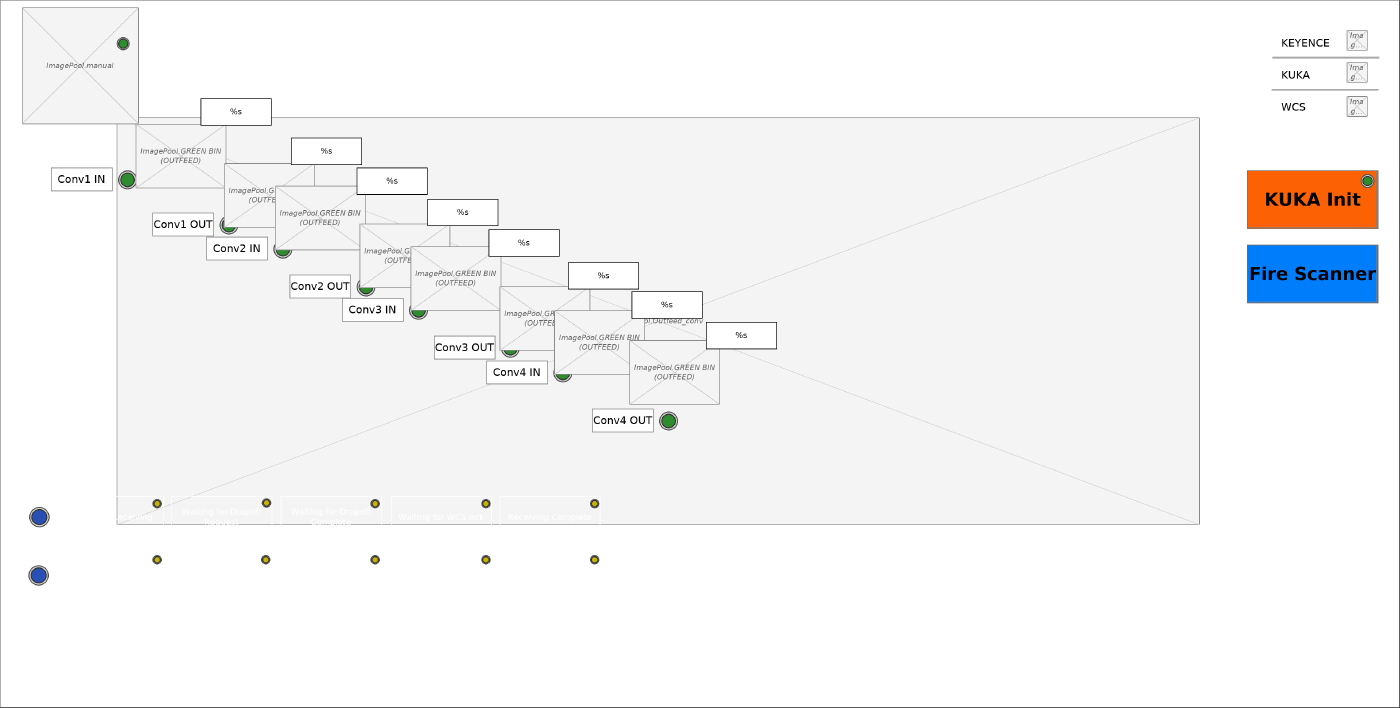
VISUALIZATION MAIN_CONTENT  // 1920x972
    Rectangle (0,0 1920x972)
    Image (160,161 1485x559), image: ImagePool.Outfeed_conv
    Group (1731,29 160x145)
        RoundedRectangle (0,0 160x145)
        RoundedRectangle (23,21 109x18), "KEYENCE"
        RoundedRectangle (23,65 92x18), "KUKA"
        RoundedRectangle (23,109 92x18), "WCS"
        Rectangle (14,49 146x2)
        Rectangle (13,93 146x2)
        Image (116,12 28x28), invisible if: IO.fbClient_QR.bConnected, image: ImagePool.no-wifi
        Image (116,12 28x28), invisible if: NOT IO.fbClient_QR.bConnected, image: ImagePool.wifi
        Image (116,56 28x28), invisible if: IO_KUKA.bPro_act, image: ImagePool.no-wifi
        Image (116,56 28x28), invisible if: NOT IO_KUKA.bPro_act, image: ImagePool.wifi
        Image (116,103 28x28), invisible if: IO.fbClient_ASRS.bConnected, image: ImagePool.no-wifi
        Image (116,103 28x28), invisible if: NOT IO.fbClient_ASRS.bConnected, image: ImagePool.wifi
    Button (1710,234 180x80), "KUKA Init", text variable: IO_KUKA.Init_Cmd
        OnMouseClick: toggle IO_KUKA.Init_Cmd
    Button (1710,336 180x80), "Fire Scanner"
        OnMouseClick: toggle IO.bRe_run_Fire
    Image (35,15 150x150), invisible if: not IO.bAutoMode, image: ImagePool.auto
    Image (30,10 160x160), invisible if: IO.bAutoMode, image: ImagePool.manual
    Group (70,230 120x32)
        RoundedRectangle (0,0 84x32), "Conv1 IN"
        Lamp1 (90,2 30x30), variable: IO.bConv1_In, style: Lamp-Lamp1-Green
    Group (209,292 127x32)
        RoundedRectangle (0,0 84x32), "Conv1 OUT"
        Lamp1 (90,2 30x30), variable: IO.bConv1_Out, style: Lamp-Lamp1-Green
    Group (283,325 120x32)
        RoundedRectangle (0,0 84x32), "Conv2 IN"
        Lamp1 (90,2 30x30), variable: IO.bConv2_In, style: Lamp-Lamp1-Green
    Group (397,377 127x32)
        RoundedRectangle (0,0 84x32), "Conv2 OUT"
        Lamp1 (90,2 30x30), variable: IO.bConv2_Out, style: Lamp-Lamp1-Green
    Group (469,409 120x32)
        RoundedRectangle (0,0 84x32), "Conv3 IN"
        Lamp1 (90,2 30x30), variable: IO.bConv3_In, style: Lamp-Lamp1-Green
    Group (595,461 127x32)
        RoundedRectangle (0,0 84x32), "Conv3 OUT"
        Lamp1 (90,2 30x30), variable: IO.bConv3_Out, style: Lamp-Lamp1-Green
    Group (667,495 120x32)
        RoundedRectangle (0,0 84x32), "Conv4 IN"
        Lamp1 (90,2 30x30), variable: IO.bConv4_In, style: Lamp-Lamp1-Green
    Group (812,561 127x32)
        RoundedRectangle (0,0 84x32), "Conv4 OUT"
        Lamp1 (90,2 30x30), variable: IO.bConv4_Out, style: Lamp-Lamp1-Green
    Lamp1 (159,50 20x20), variable: IO.bAutoMode, style: Lamp-Lamp1-Green
    Image (186,170 124x88), invisible if: IO.bBin_invi1, image: ImagePool.GREEN BIN (OUTFEED)
    Image (307,224 124x88), invisible if: IO.bBin_invi2, image: ImagePool.GREEN BIN (OUTFEED)
    Image (377,255 124x88), invisible if: IO.bBin_invi3, image: ImagePool.GREEN BIN (OUTFEED)
    Image (493,307 124x88), invisible if: IO.bBin_invi4, image: ImagePool.GREEN BIN (OUTFEED)
    Image (563,338 124x88), invisible if: IO.bBin_invi5, image: ImagePool.GREEN BIN (OUTFEED)
    Image (685,393 124x88), invisible if: IO.bBin_invi6, image: ImagePool.GREEN BIN (OUTFEED)
    Image (760,426 124x88), invisible if: IO.bBin_invi7, image: ImagePool.GREEN BIN (OUTFEED)
    Image (863,467 124x88), invisible if: IO.bBin_invi8, image: ImagePool.GREEN BIN (OUTFEED)
    RoundedRectangle (275,135 97x37), "%s", text variable: IO.abinID_Set[1]
    RoundedRectangle (399,189 97x37), "%s", text variable: IO.abinID_Set[2]
    RoundedRectangle (489,230 97x37), "%s", text variable: IO.abinID_Set[3]
    RoundedRectangle (779,360 97x37), "%s", text variable: IO.abinID_Set[6]
    RoundedRectangle (866,400 97x37), "%s", text variable: IO.abinID_Set[7]
    RoundedRectangle (586,273 97x37), "%s", text variable: IO.abinID_Set[4]
    RoundedRectangle (670,315 97x37), "%s", text variable: IO.abinID_Set[5]
    RoundedRectangle (968,442 97x37), "%s", text variable: IO.abinID_Set[8]
    Lamp1 (38,694 32x32), variable: IO_Conveyor.bReceiving_InProcess, style: Lamp-Lamp1-Blue
    Lamp1 (37,774 32x32), variable: IO_Conveyor.bEnd_InProcess, style: Lamp-Lamp1-Blue
    RoundedRectangle (235,681 138x58), "Waiting for Dropoff Request"
    RoundedRectangle (385,681 138x58), "Waiting for Dropoff Complete"
    RoundedRectangle (536,681 138x58), "Waiting for WCS Ack"
    RoundedRectangle (86,681 138x58), "Open for Receiving"
    Lamp1 (208,684 15x15), variable: IO_Conveyor.bReceiving_State_Open, style: Lamp-Lamp1-Yellow
    Lamp1 (358,683 15x15), variable: IO.bWait_dropoff_request, style: Lamp-Lamp1-Yellow
    Lamp1 (507,684 15x15), variable: IO.bWait_dropoff_complete, style: Lamp-Lamp1-Yellow
    Lamp1 (659,684 15x15), variable: IO.bWait_dropoff_ack, style: Lamp-Lamp1-Yellow
    RoundedRectangle (86,758 138x58), "Scan Complete"
    Lamp1 (208,761 15x15), variable: IO_Conveyor.bScan_Complete, style: Lamp-Lamp1-Yellow
    RoundedRectangle (235,758 138x58), "Waiting for Rack Location"
    Lamp1 (357,761 15x15), variable: IO.bWait_racklocation, style: Lamp-Lamp1-Yellow
    RoundedRectangle (385,758 138x58), "Waiting for WCS Ack"
    Lamp1 (507,761 15x15), variable: IO.bWait_WCSKUKA_ack, style: Lamp-Lamp1-Yellow
    RoundedRectangle (537,758 138x58), "Waiting for KUKA Job Complete"
    Lamp1 (659,761 15x15), variable: IO.bWait_KUKA_complete, style: Lamp-Lamp1-Yellow
    RoundedRectangle (685,681 138x58), "Receiving Complete"
    Lamp1 (808,684 15x15), variable: IO_Conveyor.bReceiving_Complete, style: Lamp-Lamp1-Yellow
    RoundedRectangle (686,758 138x58), "Waiting for WCS Ack KUKA Complete"
    Lamp1 (808,761 15x15), variable: IO.bWait_EndAck_complete, style: Lamp-Lamp1-Yellow
    Lamp1 (1865,238 21x21), variable: IO_KUKA.bPro_act, style: Lamp-Lamp1-Green
END_VISUALIZATION

(* stored: Version 1.1.0.1, ProductVersion 3.1.4024.12
   Visu MAIN_CONTENT: Id {bb272770-c777-43ab-9f80-b5de323a912d} *)
